FUNCTION_BLOCK FB_IdleState IMPLEMENTS I_State
VAR_INPUT
END_VAR
VAR_OUTPUT
END_VAR
VAR
	pConveyorSystem : POINTER TO FB_ConveyorSystem;
END_VAR

{warning 'add property implementation'}
PROPERTY Description : STRING
GET
Description := 'Idle state';
END_GET
END_PROPERTY

{warning 'add method implementation '}
METHOD DetectedPartSensor1 : BOOL
THIS^.pConveyorSystem^.SetCount();

IF NOT pConveyorSystem^.bDetectedPartSensor2 THEN
	pConveyorSystem^.SetState(pConveyorSystem^.RunningState);
END_IF
END_METHOD

{warning 'add method implementation '}
METHOD DetectedPartSensor2 : BOOL
END_METHOD

{warning 'add method implementation '}
METHOD DetectedWeightSensor : BOOL
END_METHOD

METHOD FB_init : BOOL
VAR_INPUT
	bInitRetains : BOOL; // if TRUE, the retain variables are initialized (warm start / cold start)
	bInCopyCode : BOOL;  // if TRUE, the instance afterwards gets moved into the copy code (online change)
	pConveyorSystem : POINTER TO FB_ConveyorSystem;
END_VAR
THIS^.pConveyorSystem := pConveyorSystem;
END_METHOD

{warning 'add method implementation '}
METHOD PressEmergencyStop : BOOL
pConveyorSystem^.SetState(pConveyorSystem^.EmergencyStopState);
END_METHOD

{warning 'add method implementation '}
METHOD PressStart : BOOL
END_METHOD

{warning 'add method implementation '}
METHOD PressStop : BOOL
pConveyorSystem^.SetState(pConveyorSystem^.OffState);
END_METHOD

{warning 'add method implementation '}
METHOD ProcessedWeight : BOOL
pConveyorSystem^.SetState(pConveyorSystem^.RunningState);
END_METHOD

END_FUNCTION_BLOCK

(* stored: Version 1.1.0.1, ProductVersion 3.1.4024.12
   POU FB_IdleState: Id {37e69380-dfd4-4315-bcac-08c8014fe68e}, SpecialFunc None
   Property Description: Id {6c424ffb-6e7a-4114-8585-ce0ed964f4c4}
   Get Get: Id {e9a51fd7-e525-4633-b4ab-66c38eb0d548}
   Method DetectedPartSensor1: Id {6d8df92f-c976-4b61-95fd-8239ecb732f1}
   Method DetectedPartSensor2: Id {5b909518-4bf6-4be8-a23a-d9ef40e1aa13}
   Method DetectedWeightSensor: Id {9ab55bff-01ea-4764-9ee3-8ee6818c3d6c}
   Method FB_init: Id {b554152b-4452-4073-9125-a64a14116d8e}
   Method PressEmergencyStop: Id {d260a93c-4619-4480-81aa-7564cea9291a}
   Method PressStart: Id {d4527bb4-23ac-4aa2-997c-8b0c180fa0dd}
   Method PressStop: Id {75aa1851-68d0-4d4f-af2f-6518e953291c}
   Method ProcessedWeight: Id {011bc9c1-b8a7-4e8c-9e1b-52ced7a6898c} *)
